TYPE CommandQueueMember :
STRUCT
	buffer_size				: UDINT := LibraryParameter.COMMAND_BUFFER_SIZE;
	buffer_body				: ARRAY [0..LibraryParameter.COMMAND_BUFFER_SIZE] OF DbInsertCommand;
	buffer_index			: ARRAY [0..LibraryParameter.COMMAND_BUFFER_SIZE] OF T_Arg;
	current_index			: UDINT;
	controller				: dequeue;
END_STRUCT
END_TYPE

(* stored: Version 1.1.0.1, ProductVersion 3.1.4024.12
   DUT CommandQueueMember: Id {ada4b084-8055-402d-8a7c-f4c1b53b3463} *)
